SUBAPPLICATION mapping_blink (* Subapplication Type *)
  (* Standard: 61499-2 *)
  (* Version 1.0, 2023-04-04, franz *)
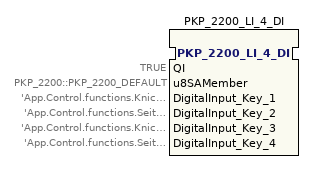
  FBS
    PKP_2200_LI_4_DI : PKP_2200_LI_4_DI(QI := TRUE, u8SAMember := PKP_2200::PKP_2200_DEFAULT, DigitalInput_Key_1 := 'App.Control.functions.Knickdeichsel_heben.IX', DigitalInput_Key_2 := 'App.Control.functions.Seitenschieber_Auf.IX', DigitalInput_Key_3 := 'App.Control.functions.Knickdeichsel_senken.IX', DigitalInput_Key_4 := 'App.Control.functions.Seitenschieber_Zu.IX');
  END_FBS
END_SUBAPPLICATION
